FUNCTION_BLOCK FB_WriteSingleRegExample
VAR
	fbMBWriteSingleReg  : FB_MBWriteSingleReg ;
	nWiteValue : INT;
	aStateMachine : (WAIT, TRIGGER, WRITE);
	fbTrigger : R_TRIG;
END_VAR

fbTrigger();
IF fbTrigger.Q THEN
	IF aStateMachine := WAIT THEN
		aStateMachine := TRIGGER;
	END_IF
END_IF
CASE aStateMachine OF
	WAIT:
		// do nothing
	TRIGGER:
	fbMBWriteSingleReg(
		sIPAddr:= , 
		nTCPPort:= , 
		nUnitID:= , 
		nMBAddr:= , 
		nValue:= TO_WORD(nWiteValue), 
		bExecute:= TRUE, 
		tTimeout:= , 
		bBusy=> , 
		bError=> , 
		nErrId=> );
		
		aStateMachine := WRITE;
	WRITE:
		// waite for response
		fbMBWriteSingleReg(bExecute := FALSE); // read until we get sth from modbus app in windows
		IF NOT fbMBWriteSingleReg.bBusy OR fbMBWriteSingleReg.bError THEN
			aStateMachine := WAIT;
		END_IF
	
END_CASE

END_FUNCTION_BLOCK

(* stored: Version 1.1.0.1, ProductVersion 3.1.4024.12
   POU FB_WriteSingleRegExample: Id {42bacbb2-5052-4ed1-a1da-659dd668a4a3}, SpecialFunc None *)
